Staubli VAL3: showItem.pgx

program showItem(string& x_sEvent[] (dimensions=1))
  local num l_nSize
  local string l_sEvent
  local num l_nKey
  local num i
  local string l_sMessage
begin
  //
  // USE this procedure to view Prog
  // that you have already saved
  //
  cls()
  call use:setView(false)
  //
  // Item list
  //
  call use:listcreate("")
  //
  l_nSize=size(saveData:sInstr)
  // refresh the list
  for i=0 to l_nSize-1
    l_sEvent=saveData:sInstr[i]
    if l_sEvent!="IF"
      call use:listadd(l_sEvent)
    endIf
  endFor
  call use:listupdate(0)
  call language:message(l_sMessage,60)
  call use:typeLen(0,13,l_sMessage,40)
  do
    l_nKey=get()
    call use:listevent(l_nKey,i,x_sEvent)
  until l_nKey==270 or l_nKey==255
  if l_nKey==255
    x_sEvent=""
  endIf
end
